PROGRAM P_Stack
VAR
	
	bCreate,bPush, bPop, bDelete : BOOL;
	pData : POINTER TO T_DATA_TYPE;
	pPush_Addr, pPop_Addr : POINTER TO T_DATA_TYPE;
	nTop : T_DATA_TYPE; 
	nIndex : ULINT;
	nSize : UDINT; 
END_VAR

P_Dynamic_Array_Stack();
P_Linked_List_Stack();


IF bCreate AND (pData = 0) THEN 
	nSize := SIZEOF(T_DATA_TYPE)*10;
	pData := __NEW(T_DATA_TYPE,nSize);
	bCreate := FALSE;
	END_IF

IF bPush THEN 
	pData[nIndex] := nIndex + 10;
	nTop := pData[nIndex];
	pPush_Addr := ADR(pData[nIndex]);
	nIndex := nIndex + 1;
	bPush := FALSE;
	END_IF

IF bPop AND (nIndex > 0) THEN 
	nIndex := nIndex - 1;
	nTop := pData[nIndex];
	pPop_Addr := ADR(pData[nIndex]);
	bPop := FALSE;
	END_IF
	
IF bDelete THEN 
	__DELETE(pData);
	bDelete := FALSE;
	END_IF

END_PROGRAM

(* stored: Version 1.1.0.1, ProductVersion 3.1.4024.4
   POU P_Stack: Id {6d895120-20ec-4ebe-b215-006e9cde9ef5}, SpecialFunc None *)
